Staubli VAL3: read_data.pgx

public program read_data()
  local string sInputData_1
  local num nRec
  local num nReceived
  local num nInputData_1
begin

  putln("Start to read data !")

  do
    sInputData_1 = ""
    do
      nReceived=sioGet(sioASCII,nRec)
      sInputData_1 = sInputData_1 + chr(nRec)

    until nRec == 13 or nReceived == -1

    if nReceived != 1
      check_status = false
      stopMove()
      cls()
      putln("Communication error !")
      disablePower()
    endIf

    toNum(sInputData_1 , nInputData_1, check_status)

    //put("Reference Velocity [mm/s]: ")
    //put(nInputData_1)
    //putln("")



    if getMoveId() >= 0.1
       Ref_Vel = nInputData_1
    elseIf getMoveId() < 0.1
       Ref_Vel = print_vel
    endIf

   // putln(Ref_Vel)


   //delay(0.001)

  until check_status != true

end
